PROGRAM P_AbstractFactory
VAR
    fbDatabaseLoggerFactory  : FB_DatabaseLoggerFactory('MyDatabase', 'User', 'Password');
    refDatabaseLoggerFactory : REFERENCE TO FB_DatabaseLoggerFactory := fbDatabaseLoggerFactory;
    fbLogger                 : FB_Logger(refDatabaseLoggerFactory);	
    sRetMsg                  : STRING;
END_VAR

sRetMsg := fbLogger.Write('Hello');

END_PROGRAM

(* stored: Version 1.1.0.1, ProductVersion 3.1.4024.12
   POU P_AbstractFactory: Id {fd6e49ae-9c60-4ba4-ba01-45f20a4b6c2c}, SpecialFunc None *)
